// TwinCAT 3 PLC project Untitled1
// ProgramVersion: 3.1.4024.0
// libraries:
//   Tc2_Standard, * (Beckhoff Automation GmbH)
//   Tc2_System, * (Beckhoff Automation GmbH)
//   Tc3_Module, * (Beckhoff Automation GmbH)
// project tree:
//   GVLs/ GVL.TcGVL
//   / PlcTask.TcTTO, Task_Koffie.TcTTO, Task_Reis.TcTTO
//   POUs/ fBoolToText.TcPOU, MAIN.TcPOU, PGR_Koffie.TcPOU, PRg_Reis.TcPOU
// real-time tasks:
//   TASK PlcTask: cycle T#10ms, priority 20, ADS port 350
//   TASK Task_Reis: cycle T#10ms, priority 21, ADS port 351
//   TASK Task_Koffie: cycle T#10ms, priority 22, ADS port 352

CONFIGURATION Untitled1
    RESOURCE PLC ON TwinCAT3
        TASK PlcTask(INTERVAL := T#10ms, PRIORITY := 20);
        TASK Task_Koffie(INTERVAL := T#10ms, PRIORITY := 22);
        TASK Task_Reis(INTERVAL := T#10ms, PRIORITY := 21);
        PROGRAM MAIN WITH PlcTask : MAIN;
        PROGRAM PGR_Koffie WITH Task_Koffie : PGR_Koffie;
        PROGRAM PRg_Reis WITH Task_Reis : PRg_Reis;
    END_RESOURCE
END_CONFIGURATION

// ---- GVLs/GVL.TcGVL

VAR_GLOBAL
    bVraagKoffie  : BOOL;
    bKoffieGereed : BOOL;
END_VAR

// ---- POUs/MAIN.TcPOU
PROGRAM MAIN
VAR
END_VAR

END_PROGRAM

// ---- POUs/PGR_Koffie.TcPOU
PROGRAM PGR_Koffie
VAR_EXTERNAL
    bVraagKoffie  : BOOL;
    bKoffieGereed : BOOL;
END_VAR

VAR
    tKoffie : TON;
    sStatus : STRING[50];
	 iState : INT; // 0=Idle, 1=KoffieZetten, 2=Klaar
	tReis: Ton;
END_VAR

CASE iState OF

    0: // Idle
        sStatus := 'Geen koffie opdracht';
        tKoffie(IN := FALSE);
        IF bVraagKoffie THEN
            iState := 1;
        END_IF

    1: // Koffie zetten
        sStatus := 'Koffie wordt gezet';
        tKoffie(IN := TRUE, PT := T#3s);
        IF tKoffie.Q THEN
            tKoffie(IN := FALSE);
            bKoffieGereed := TRUE;
            bVraagKoffie := FALSE;
            iState := 2;
        END_IF

    2: // Klaar
        sStatus := 'Koffie is klaar';

END_CASE

END_PROGRAM

// ---- POUs/PRg_Reis.TcPOU
PROGRAM PRg_Reis
VAR_EXTERNAL
    bVraagKoffie  : BOOL;
    bKoffieGereed : BOOL;
END_VAR

VAR
    tReis : TON;
    sStatus : STRING[50];
    bAangekomen : BOOL;
	iState: INT;// 0=Idle, 1=Reizen, 2=Aangekomen, 3=WachtenOpKoffie
	tKoffie: Ton;
END_VAR

CASE iState OF

    0: // Idle
        sStatus := 'Start reis';
        tReis(IN := FALSE);
        iState := 1;

    1: // Reizen
        sStatus := 'Onderweg naar Deventer';
        tReis(IN := TRUE, PT := T#5s);
        IF tReis.Q THEN
            tReis(IN := FALSE);
            bVraagKoffie := TRUE;
            iState := 2;
        END_IF

    2: // Aangekomen
        sStatus := 'Aangekomen in Deventer';
        iState := 3;

    3: // Wachten op koffie
        sStatus := 'Wachten op koffie';
        IF bKoffieGereed THEN
            sStatus := 'Koffie ontvangen, verder reizen';
        END_IF

END_CASE

END_PROGRAM

// ---- POUs/fBoolToText.TcPOU
FUNCTION fBoolToText  : STRING
VAR_INPUT
    bValue : BOOL;
END_VAR

IF bValue THEN
    fBoolToText := 'TRUE';
ELSE
    fBoolToText := 'FALSE';
END_IF

END_FUNCTION
